FUNCTION_BLOCK Switch_2P
VAR_INPUT
END_VAR
VAR_OUTPUT
END_VAR
VAR
	DI_Input at %I* : bool;
END_VAR

PROPERTY position0 : BOOL
GET
position0 := not Switch_2P;
END_GET
END_PROPERTY

PROPERTY position1 : BOOL
GET
position1 := Switch_2P;
END_GET
END_PROPERTY

END_FUNCTION_BLOCK

(* stored: Version 1.1.0.1
   POU Switch_2P: Id {1844778d-91ff-4d36-98a4-04da56985296}, SpecialFunc None
   Property position0: Id {f2d4dead-14cd-458e-901d-9a307c79e61a}
   Get Get: Id {2f12a057-fcc5-4a70-a53e-bc0a04fc1234}
   Property position1: Id {39c309c0-e723-4261-b29b-4af7e289ee5a}
   Get Get: Id {1a260927-d8ec-49aa-a2f8-cec52816d6c4} *)
